Universal Robots PolyScope program: barriere.urp

Program barriere (installation=barriere directory=/home/ur/ursim/ursim-5.11.0.108249/programs/Bbraun createdIn=5.11.0.108249 lastSavedIn=5.11.0.108249 robotSerialNumber=20195299999)
Calibrated DH parameters: a=[0, -0.6127, -0.57155, 0, 0, 0]; d=[0.1807, 0, 0, 0.17415, 0.11985, 0.11655]; alpha=[1.570796, 0, 0, 1.570796, -1.570796, 0]; deltaTheta=[0, 0, 0, 0, 0, 0]
BeforeStart
  MoveJ speed 60 deg/s, acceleration 80 deg/s^2 (useActiveTCP=true) feature=Base
    Waypoint Waypoint_2 (Relative): relativeFromPosition TCP in base x=350.519 y=-609.706 z=727.359 mm, rx=-0.033 ry=-2.2098 rz=2.203 rad; joints [-37.661, -93.735, -105.069, 18.5, 35.948, 0.246] deg; TCP in base x=350.519 y=-609.706 z=727.359 mm, rx=-0.033 ry=-2.2098 rz=2.203 rad; joints [-37.661, -93.735, -105.069, 18.5, 35.948, 0.246] deg
Robot Program (runOnlyOnce=false)
  MoveJ speed 60 deg/s, acceleration 80 deg/s^2 (useActiveTCP=true) feature=Base
    Waypoint machine: TCP in base x=624.789 y=141.965 z=977.916 mm, rx=1.1895 ry=0.1776 rz=1.7043 rad; joints [37.215, -96.29, -77.9, 47.486, 38.928, 179.779] deg
    Waypoint magasin: TCP in base x=549.946 y=-670.02 z=977.916 mm, rx=1.1895 ry=0.1776 rz=1.7043 rad; joints [-40.625, -114.195, -58.078, 23.237, 101.728, 232.953] deg
